(* CODESYS project Soru_6.project
   Title: Adsız2
   Version: 0.0.0.0
   Author: Enes

Project tree, tasks and I/O mapping:
  MyController : TM241C24T/U, Schneider Electric, order no. TM241C24T/U, version 4.0.6.18
    application Application
      task MAST (cyclic, interval 20 ms, priority 15, watchdog 100 ms x 1) calls POU
      global variables GVL
      program POU [LD]
    DI : Digital Inputs, Schneider Electric, version 4.0.6.18
        input  iwDI_IW0 : WORD  // IW0
        input  ibDI_IB1 : BYTE  // IB1
    DQ : Digital Outputs, Schneider Electric, version 4.0.6.18
        output qwDQ_QW0 : WORD  // QW0
        output qbDQ_QB1 : BYTE  // QB1
    Counters : Counters, Schneider Electric, version 4.0.6.18
    Pulse_Generators : Pulse Generators, Schneider Electric, version 4.0.6.18
    Cartridge_1 : Cartridge, Schneider Electric, version 4.0.6.18
    IO_Bus : IO bus - TM3, Schneider Electric, version 4.0.6.18
    COM_Bus : COM bus, Schneider Electric, version 4.0.6.18
    Serial_Line_1 : Serial line, Schneider Electric, version 4.0.6.18
      SoMachine_Network_Manager : SoMachine-Network Manager, Schneider Electric, version 4.0.0.2
    Serial_Line_2 : Serial line, Schneider Electric, version 4.0.6.18
      Modbus_Manager : Modbus Manager, Schneider Electric, version 4.0.0.2
*)

// MyController/Application/GVL
VAR_GLOBAL
END_VAR

// MyController/Application/POU
PROGRAM POU
VAR
	Start: BOOL;
	Stop: BOOL;
	M0: BOOL;
	Q3: BOOL;
	Q2: BOOL;
	S3: BOOL;
	T37: TON;
	S2: BOOL;
	Q1: BOOL;
	T38: TON;
	S1: BOOL;
	M1: BOOL;
END_VAR
VAR // added by the converter: edge detectors and wires of the graphical bodies
    _w1, _w2 : BOOL;
END_VAR

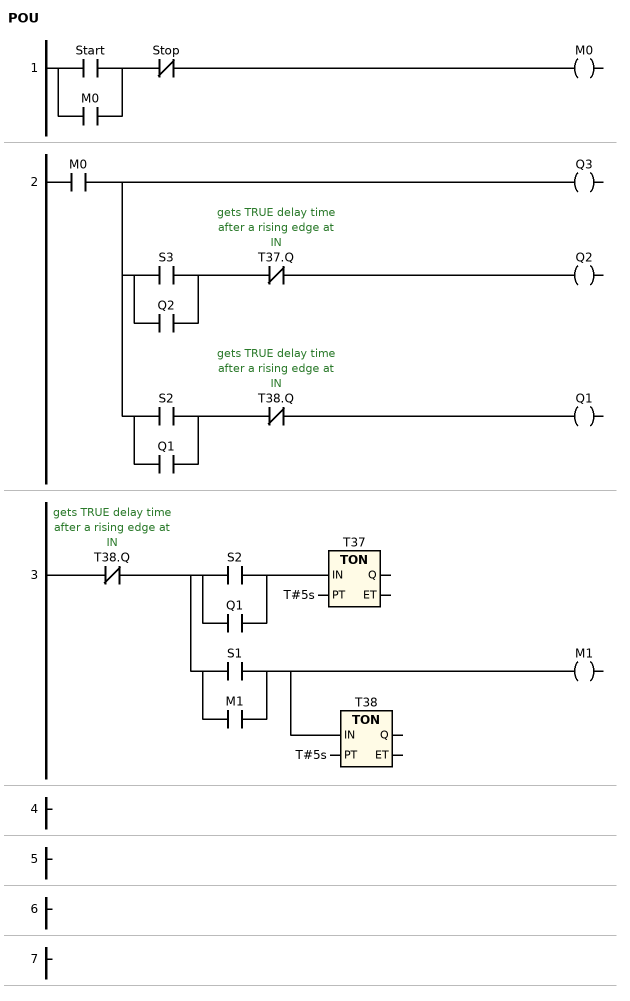
// NETWORK 1
M0 := (Start OR M0) AND NOT Stop;

// NETWORK 2
//   T37.Q: gets TRUE delay time after a rising edge at IN
//   T38.Q: gets TRUE delay time after a rising edge at IN
Q3 := M0;
Q2 := M0 AND (S3 OR Q2) AND NOT T37.Q;
Q1 := M0 AND (S2 OR Q1) AND NOT T38.Q;

// NETWORK 3
//   T38.Q: gets TRUE delay time after a rising edge at IN
_w1 := NOT T38.Q;
T37(IN := _w1 AND (S2 OR Q1), PT := T#5s); // TON
_w2 := _w1 AND (S1 OR M1);
M1 := _w2;
T38(IN := _w2, PT := T#5s); // TON

// NETWORK 4

// NETWORK 5

// NETWORK 6

// NETWORK 7

END_PROGRAM
